FUNCTION_BLOCK T_CountReturnsCorrect EXTENDS T_UnitTestBase
VAR
  list : T_ComponentsCollection(10);
  newComponent : ARRAY [1..5] OF T_Component;
  expected, actual : UINT;
  result : BOOL;
END_VAR

list.AddComponent(newComponent[1]);
list.AddComponent(newComponent[2]);
list.AddComponent(newComponent[3]);
list.AddComponent(newComponent[4]);

expected := 4;
actual := list.Count;

assertion.AssertEquals_UINT(expected, actual, 'actual := list.Count');
TestFinished();

END_FUNCTION_BLOCK

(* stored: Version 1.1.0.1, ProductVersion 3.1.4024.12
   POU T_CountReturnsCorrect: Id {e60208ed-9066-4494-9717-1e67b98003a8}, SpecialFunc None *)
